LIN {X 0,Y 76.408,Z 663.728,A -85,B 0,C 180,E1 -30054.723,E2 -30054.723} C_VEL
LIN {X 0,Y 91.454,Z 656.934,A -85,B 0,C 180,E1 -30057.454,E2 -30057.454} C_VEL
LIN {X 0,Y 105.427,Z 649.252,A -85,B 0,C 180,E1 -30059.333,E2 -30059.333} C_VEL
LIN {X 0,Y 119.484,Z 640.09,A -85,B 0,C 180,E1 -30060.705,E2 -30060.705} C_VEL
LIN {X 0,Y 122.579,Z 641.733,A -85,B 0,C 180,E1 -30060.957,E2 -30060.957} C_VEL
LIN {X 0,Y 122.579,Z 670.572,A -85,B 0,C 180,E1 -30060.957,E2 -30060.957} C_VEL
LIN {X 0,Y 87.271,Z 670.572,A -85,B 0,C 180,E1 -30060.555,E2 -30060.555} C_VEL
LIN {X 0,Y 85.271,Z 668.572,A -85,B 0,C 180,E1 -30060.522,E2 -30060.522} C_VEL
LIN {X 0,Y 85.271,Z 662.674,A -85,B 0,C 180,E1 -30060.522,E2 -30060.522} C_VEL
LIN {X 0,Y 82.621,Z 660.817,A -85,B 0,C 180,E1 -30061.003,E2 -30061.003} C_VEL
LIN {X 0,Y 66.904,Z 666.82,A -85,B 0,C 180,E1 -30063.683,E2 -30063.683} C_VEL
LIN {X 0,Y 50.83,Z 671.566,A -85,B 0,C 180,E1 -30067.949,E2 -30067.949} C_VEL
LIN {X 0,Y 36.351,Z 674.72,A -85,B 0,C 180,E1 -30074.829,E2 -30074.829} C_VEL
LIN {X 0,Y 23.869,Z 676.592,A -85,B 0,C 180,E1 -30087.954,E2 -30087.954} C_VEL
LIN {X 0,Y 14.482,Z 677.517,A -85,B 0,C 180,E1 -30120.968,E2 -30120.968} C_VEL
LIN {X 0,Y 13.026,Z 677.662,A -85,B 0,C 180,E1 -30149.999,E2 -30149.999} C_VEL
LIN {X 0,Y 18.476,Z 677.182,A -85,B 0,C 180,E1 -30199.529,E2 -30199.529} C_VEL
LIN {X 0,Y 29.902,Z 675.859,A -85,B 0,C 180,E1 -30220.071,E2 -30220.071} C_VEL
LIN {X 0,Y 42.962,Z 673.47,A -85,B 0,C 180,E1 -30228.96,E2 -30228.96} C_VEL
LIN {X 0,Y 56.549,Z 670.165,A -85,B 0,C 180,E1 -30233.85,E2 -30233.85} C_VEL
LIN {X 0,Y 73.854,Z 664.481,A -85,B 0,C 180,E1 -30237.674,E2 -30237.674} C_VEL
LIN {X 0,Y 82.255,Z 661.114,A -85,B 0,C 180,E1 -30239.018,E2 -30239.018} C_VEL
LIN {X 0,Y 66.784,Z 667.102,A -85,B 0,C 180,E1 -30241.359,E2 -30241.359} C_VEL
LIN {X 0,Y 56.339,Z 670.446,A -85,B 0,C 180,E1 -30243.672,E2 -30243.672} C_VEL
LIN {X 0,Y 38.702,Z 674.763,A -85,B 0,C 180,E1 -30250.461,E2 -30250.461} C_VEL
LIN {X 0,Y 29.453,Z 676.412,A -85,B 0,C 180,E1 -30257.362,E2 -30257.362} C_VEL
LIN {X 0,Y 17.865,Z 677.853,A -85,B 0,C 180,E1 -30278.115,E2 -30278.115} C_VEL
LIN {X 0,Y 12.75,Z 678.415,A -85,B 0,C 180,E1 -30330.001,E2 -30330.001} C_VEL
LIN {X 0,Y 17.865,Z 677.831,A -85,B 0,C 180,E1 -30381.889,E2 -30381.889} C_VEL
LIN {X 0,Y 29.453,Z 676.367,A -85,B 0,C 180,E1 -30402.642,E2 -30402.642} C_VEL
LIN {X 0,Y 42.634,Z 673.826,A -85,B 0,C 180,E1 -30411.517,E2 -30411.517} C_VEL
LIN {X 0,Y 59.812,Z 669.269,A -85,B 0,C 180,E1 -30417.155,E2 -30417.155} C_VEL
LIN {X 0,Y 75.194,Z 663.882,A -85,B 0,C 180,E1 -30420.001,E2 -30420.001} C_VEL
LIN {X 0,Y 82.621,Z 660.817,A -85,B 0,C 180,E1 -30421.003,E2 -30421.003} C_VEL
LIN {X 0,Y 85.355,Z 662.662,A -85,B 0,C 180,E1 -30421.312,E2 -30421.312} C_VEL
LIN {X 0,Y 85.355,Z 683.352,A -85,B 0,C 180,E1 -30421.312,E2 -30421.312} C_VEL
LIN {X 0,Y 46.513,Z 683.352,A -85,B 0,C 180,E1 -30420.995,E2 -30420.995} C_VEL
LIN {X 0,Y 44.513,Z 681.352,A -85,B 0,C 180,E1 -30420.964,E2 -30420.964} C_VEL
LIN {X 0,Y 44.513,Z 675.576,A -85,B 0,C 180,E1 -30420.964,E2 -30420.964} C_VEL
LIN {X 0,Y 42.182,Z 673.61,A -85,B 0,C 180,E1 -30421.494,E2 -30421.494} C_VEL
LIN {X 0,Y 28.281,Z 676.02,A -85,B 0,C 180,E1 -30426.261,E2 -30426.261} C_VEL
LIN {X 0,Y 14.872,Z 677.367,A -85,B 0,C 180,E1 -30439.067,E2 -30439.067} C_VEL
LIN {X 0,Y 5.933,Z 677.87,A -85,B 0,C 180,E1 -30509.997,E2 -30509.997} C_VEL
LIN {X 0,Y 14.869,Z 677.39,A -85,B 0,C 180,E1 -30580.964,E2 -30580.964} C_VEL
LIN {X 0,Y 28.275,Z 676.067,A -85,B 0,C 180,E1 -30593.829,E2 -30593.829} C_VEL
LIN {X 0,Y 42.177,Z 673.683,A -85,B 0,C 180,E1 -30598.76,E2 -30598.76} C_VEL
LIN {X 0,Y 28.156,Z 676.202,A -85,B 0,C 180,E1 -30603.224,E2 -30603.224} C_VEL
LIN {X 0,Y 14.571,Z 677.643,A -85,B 0,C 180,E1 -30615.289,E2 -30615.289} C_VEL
LIN {X 0,Y 5.636,Z 678.207,A -85,B 0,C 180,E1 -30690.003,E2 -30690.003} C_VEL
LIN {X 0,Y 14.572,Z 677.621,A -85,B 0,C 180,E1 -30764.717,E2 -30764.717} C_VEL
LIN {X 0,Y 28.157,Z 676.157,A -85,B 0,C 180,E1 -30776.78,E2 -30776.78} C_VEL
LIN {X 0,Y 42.182,Z 673.61,A -85,B 0,C 180,E1 -30781.494,E2 -30781.494} C_VEL
LIN {X 0,Y 42.182,Z 673.61,A -85,B 0,C 180,E1 -30781.494,E2 -30781.494}

QRS_NEXT_CUT()

QRS_NEXT()
QRS_HOME()

END
